PROGRAM P_Demo_UInt64And
VAR
    uliStatus    : T_ULARGE_INTEGER;; // 状态寄存器（64 位）
    uliMask      : T_ULARGE_INTEGER;; // 掩码：低 16 位
    uliFaultCode : T_ULARGE_INTEGER;; // 屏蔽后的故障码
    bMaskNow     : BOOL;; // 触发屏蔽
END_VAR

// ============================================================
// Tc2_Utilities.UInt64And 演示程序（FUNCTION，单周期触发）
// ============================================================
// 场景：ADS Raw 报文里把状态寄存器的 64 位状态位按掩码取出特定子位段（如故障码低 16 位）。
// 价值：替代分别 AND 高低 DWORD 两行；语义更清晰。
// 验证步骤：
//   1. 把本 PROGRAM 加到 PlcTask 调用列表
//   2. 编译 + 登录
//   3. 在线把 b... 触发位置 TRUE 一个周期
//   4. 观察输出变量是否符合期望
// ============================================================

uliMask := ULARGE_INTEGER(0, 16#0000FFFF);   // 取低 16 位的掩码
IF bMaskNow THEN
    uliFaultCode := UInt64And(uliStatus, uliMask);
    bMaskNow := FALSE;
END_IF;

END_PROGRAM

(* stored: Version 1.1.0.1, ProductVersion 3.1.4024.5
   POU P_Demo_UInt64And: Id {a71ee21b-b323-5540-a0b2-7a84dbff00e1}, SpecialFunc None *)
